    report_progress()
    set_digital_out(0, False)
    new_pose = pose_trans(tuft_coords, p[1.0096, 0.7853, 0.1500, 0, 0, 0])
    movel(p[new_pose[0], new_pose[1], new_pose[2], current_pose[3], current_pose[4], current_pose[5]], a=0.8, v=0.2000)
    report_progress()
    new_pose = pose_trans(tuft_coords, p[1.0115, 0.2667, 0.1500, 0, 0, 0])
    movel(p[new_pose[0], new_pose[1], new_pose[2], current_pose[3], current_pose[4], current_pose[5]], a=1.2, v=0.2000)
    report_progress()
    new_pose = pose_trans(tuft_coords, p[1.0115, 0.2667, -0.0020, 0, 0, 0])
    movel(p[new_pose[0], new_pose[1], new_pose[2], current_pose[3], current_pose[4], current_pose[5]], a=0.8, v=0.2000)
    report_progress()
    set_digital_out(0, True)
    new_pose = pose_trans(tuft_coords, p[1.0115, 0.7833, -0.0020, 0, 0, 0])
    movel(p[new_pose[0], new_pose[1], new_pose[2], current_pose[3], current_pose[4], current_pose[5]], a=1.2, v=0.0600)
    report_progress()
    set_digital_out(0, False)
    new_pose = pose_trans(tuft_coords, p[1.0115, 0.7833, 0.1500, 0, 0, 0])
    movel(p[new_pose[0], new_pose[1], new_pose[2], current_pose[3], current_pose[4], current_pose[5]], a=0.8, v=0.2000)
    report_progress()
    new_pose = pose_trans(tuft_coords, p[1.0135, 0.2687, 0.1500, 0, 0, 0])
    movel(p[new_pose[0], new_pose[1], new_pose[2], current_pose[3], current_pose[4], current_pose[5]], a=1.2, v=0.2000)
    report_progress()
    new_pose = pose_trans(tuft_coords, p[1.0135, 0.2687, -0.0020, 0, 0, 0])
    movel(p[new_pose[0], new_pose[1], new_pose[2], current_pose[3], current_pose[4], current_pose[5]], a=0.8, v=0.2000)
    report_progress()
    set_digital_out(0, True)
    new_pose = pose_trans(tuft_coords, p[1.0135, 0.7813, -0.0020, 0, 0, 0])
    movel(p[new_pose[0], new_pose[1], new_pose[2], current_pose[3], current_pose[4], current_pose[5]], a=1.2, v=0.0600)
    report_progress()
    set_digital_out(0, False)
    new_pose = pose_trans(tuft_coords, p[1.0135, 0.7813, 0.1500, 0, 0, 0])
    movel(p[new_pose[0], new_pose[1], new_pose[2], current_pose[3], current_pose[4], current_pose[5]], a=0.8, v=0.2000)
    report_progress()
    new_pose = pose_trans(tuft_coords, p[1.0154, 0.2707, 0.1500, 0, 0, 0])
    movel(p[new_pose[0], new_pose[1], new_pose[2], current_pose[3], current_pose[4], current_pose[5]], a=1.2, v=0.2000)
    report_progress()
    new_pose = pose_trans(tuft_coords, p[1.0154, 0.2707, -0.0020, 0, 0, 0])
    movel(p[new_pose[0], new_pose[1], new_pose[2], current_pose[3], current_pose[4], current_pose[5]], a=0.8, v=0.2000)
    report_progress()
    set_digital_out(0, True)
    new_pose = pose_trans(tuft_coords, p[1.0154, 0.7793, -0.0020, 0, 0, 0])
    movel(p[new_pose[0], new_pose[1], new_pose[2], current_pose[3], current_pose[4], current_pose[5]], a=1.2, v=0.0600)
    report_progress()
    set_digital_out(0, False)
    new_pose = pose_trans(tuft_coords, p[1.0154, 0.7793, 0.1500, 0, 0, 0])
    movel(p[new_pose[0], new_pose[1], new_pose[2], current_pose[3], current_pose[4], current_pose[5]], a=0.8, v=0.2000)
    report_progress()
    new_pose = pose_trans(tuft_coords, p[1.0174, 0.2727, 0.1500, 0, 0, 0])
    movel(p[new_pose[0], new_pose[1], new_pose[2], current_pose[3], current_pose[4], current_pose[5]], a=1.2, v=0.2000)
    report_progress()
    new_pose = pose_trans(tuft_coords, p[1.0174, 0.2727, -0.0020, 0, 0, 0])
    movel(p[new_pose[0], new_pose[1], new_pose[2], current_pose[3], current_pose[4], current_pose[5]], a=0.8, v=0.2000)
    report_progress()
    set_digital_out(0, True)
    new_pose = pose_trans(tuft_coords, p[1.0174, 0.7773, -0.0020, 0, 0, 0])
    movel(p[new_pose[0], new_pose[1], new_pose[2], current_pose[3], current_pose[4], current_pose[5]], a=1.2, v=0.0600)
    report_progress()
    set_digital_out(0, False)
    new_pose = pose_trans(tuft_coords, p[1.0174, 0.7773, 0.1500, 0, 0, 0])
    movel(p[new_pose[0], new_pose[1], new_pose[2], current_pose[3], current_pose[4], current_pose[5]], a=0.8, v=0.2000)
    report_progress()
    new_pose = pose_trans(tuft_coords, p[1.0193, 0.2746, 0.1500, 0, 0, 0])
    movel(p[new_pose[0], new_pose[1], new_pose[2], current_pose[3], current_pose[4], current_pose[5]], a=1.2, v=0.2000)
    report_progress()
    new_pose = pose_trans(tuft_coords, p[1.0193, 0.2746, -0.0020, 0, 0, 0])
    movel(p[new_pose[0], new_pose[1], new_pose[2], current_pose[3], current_pose[4], current_pose[5]], a=0.8, v=0.2000)
    report_progress()
    set_digital_out(0, True)
    new_pose = pose_trans(tuft_coords, p[1.0193, 0.7754, -0.0020, 0, 0, 0])
    movel(p[new_pose[0], new_pose[1], new_pose[2], current_pose[3], current_pose[4], current_pose[5]], a=1.2, v=0.0600)
    report_progress()
    set_digital_out(0, False)
    new_pose = pose_trans(tuft_coords, p[1.0193, 0.7754, 0.1500, 0, 0, 0])
    movel(p[new_pose[0], new_pose[1], new_pose[2], current_pose[3], current_pose[4], current_pose[5]], a=0.8, v=0.2000)
    report_progress()
    new_pose = pose_trans(tuft_coords, p[1.0212, 0.2766, 0.1500, 0, 0, 0])
    movel(p[new_pose[0], new_pose[1], new_pose[2], current_pose[3], current_pose[4], current_pose[5]], a=1.2, v=0.2000)
    report_progress()
    new_pose = pose_trans(tuft_coords, p[1.0212, 0.2766, -0.0020, 0, 0, 0])
    movel(p[new_pose[0], new_pose[1], new_pose[2], current_pose[3], current_pose[4], current_pose[5]], a=0.8, v=0.2000)
    report_progress()
    set_digital_out(0, True)
    new_pose = pose_trans(tuft_coords, p[1.0212, 0.7734, -0.0020, 0, 0, 0])
    movel(p[new_pose[0], new_pose[1], new_pose[2], current_pose[3], current_pose[4], current_pose[5]], a=1.2, v=0.0600)
    report_progress()
    set_digital_out(0, False)
    new_pose = pose_trans(tuft_coords, p[1.0212, 0.7734, 0.1500, 0, 0, 0])
    movel(p[new_pose[0], new_pose[1], new_pose[2], current_pose[3], current_pose[4], current_pose[5]], a=0.8, v=0.2000)
    report_progress()
    new_pose = pose_trans(tuft_coords, p[1.0232, 0.2786, 0.1500, 0, 0, 0])
    movel(p[new_pose[0], new_pose[1], new_pose[2], current_pose[3], current_pose[4], current_pose[5]], a=1.2, v=0.2000)
    report_progress()
    new_pose = pose_trans(tuft_coords, p[1.0232, 0.2786, -0.0020, 0, 0, 0])
    movel(p[new_pose[0], new_pose[1], new_pose[2], current_pose[3], current_pose[4], current_pose[5]], a=0.8, v=0.2000)
    report_progress()
    set_digital_out(0, True)
    new_pose = pose_trans(tuft_coords, p[1.0232, 0.7714, -0.0020, 0, 0, 0])
    movel(p[new_pose[0], new_pose[1], new_pose[2], current_pose[3], current_pose[4], current_pose[5]], a=1.2, v=0.0600)
    report_progress()
    set_digital_out(0, False)
    new_pose = pose_trans(tuft_coords, p[1.0232, 0.7714, 0.1500, 0, 0, 0])
    movel(p[new_pose[0], new_pose[1], new_pose[2], current_pose[3], current_pose[4], current_pose[5]], a=0.8, v=0.2000)
    report_progress()
    new_pose = pose_trans(tuft_coords, p[1.0251, 0.2826, 0.1500, 0, 0, 0])
    movel(p[new_pose[0], new_pose[1], new_pose[2], current_pose[3], current_pose[4], current_pose[5]], a=1.2, v=0.2000)
    report_progress()
    new_pose = pose_trans(tuft_coords, p[1.0251, 0.2826, -0.0020, 0, 0, 0])
    movel(p[new_pose[0], new_pose[1], new_pose[2], current_pose[3], current_pose[4], current_pose[5]], a=0.8, v=0.2000)
    report_progress()
    set_digital_out(0, True)
    new_pose = pose_trans(tuft_coords, p[1.0251, 0.7674, -0.0020, 0, 0, 0])
    movel(p[new_pose[0], new_pose[1], new_pose[2], current_pose[3], current_pose[4], current_pose[5]], a=1.2, v=0.0600)
    report_progress()
    set_digital_out(0, False)
    new_pose = pose_trans(tuft_coords, p[1.0251, 0.7674, 0.1500, 0, 0, 0])
    movel(p[new_pose[0], new_pose[1], new_pose[2], current_pose[3], current_pose[4], current_pose[5]], a=0.8, v=0.2000)
    report_progress()
    new_pose = pose_trans(tuft_coords, p[1.0271, 0.2845, 0.1500, 0, 0, 0])
    movel(p[new_pose[0], new_pose[1], new_pose[2], current_pose[3], current_pose[4], current_pose[5]], a=1.2, v=0.2000)
    report_progress()
    new_pose = pose_trans(tuft_coords, p[1.0271, 0.2845, -0.0020, 0, 0, 0])
    movel(p[new_pose[0], new_pose[1], new_pose[2], current_pose[3], current_pose[4], current_pose[5]], a=0.8, v=0.2000)
    report_progress()
    set_digital_out(0, True)
    new_pose = pose_trans(tuft_coords, p[1.0271, 0.7655, -0.0020, 0, 0, 0])
    movel(p[new_pose[0], new_pose[1], new_pose[2], current_pose[3], current_pose[4], current_pose[5]], a=1.2, v=0.0600)
    report_progress()
    set_digital_out(0, False)
    new_pose = pose_trans(tuft_coords, p[1.0271, 0.7655, 0.1500, 0, 0, 0])
    movel(p[new_pose[0], new_pose[1], new_pose[2], current_pose[3], current_pose[4], current_pose[5]], a=0.8, v=0.2000)
    report_progress()
    new_pose = pose_trans(tuft_coords, p[1.0290, 0.2865, 0.1500, 0, 0, 0])
    movel(p[new_pose[0], new_pose[1], new_pose[2], current_pose[3], current_pose[4], current_pose[5]], a=1.2, v=0.2000)
    report_progress()
    new_pose = pose_trans(tuft_coords, p[1.0290, 0.2865, -0.0020, 0, 0, 0])
    movel(p[new_pose[0], new_pose[1], new_pose[2], current_pose[3], current_pose[4], current_pose[5]], a=0.8, v=0.2000)
    report_progress()
    set_digital_out(0, True)
    new_pose = pose_trans(tuft_coords, p[1.0290, 0.7635, -0.0020, 0, 0, 0])
    movel(p[new_pose[0], new_pose[1], new_pose[2], current_pose[3], current_pose[4], current_pose[5]], a=1.2, v=0.0600)
    report_progress()
    set_digital_out(0, False)
    new_pose = pose_trans(tuft_coords, p[1.0290, 0.7635, 0.1500, 0, 0, 0])
    movel(p[new_pose[0], new_pose[1], new_pose[2], current_pose[3], current_pose[4], current_pose[5]], a=0.8, v=0.2000)
    report_progress()
    new_pose = pose_trans(tuft_coords, p[1.0310, 0.2885, 0.1500, 0, 0, 0])
    movel(p[new_pose[0], new_pose[1], new_pose[2], current_pose[3], current_pose[4], current_pose[5]], a=1.2, v=0.2000)
    report_progress()
    new_pose = pose_trans(tuft_coords, p[1.0310, 0.2885, -0.0020, 0, 0, 0])
    movel(p[new_pose[0], new_pose[1], new_pose[2], current_pose[3], current_pose[4], current_pose[5]], a=0.8, v=0.2000)
    report_progress()
    set_digital_out(0, True)
    new_pose = pose_trans(tuft_coords, p[1.0310, 0.7615, -0.0020, 0, 0, 0])
    movel(p[new_pose[0], new_pose[1], new_pose[2], current_pose[3], current_pose[4], current_pose[5]], a=1.2, v=0.0600)
    report_progress()
    set_digital_out(0, False)
    new_pose = pose_trans(tuft_coords, p[1.0310, 0.7615, 0.1500, 0, 0, 0])
    movel(p[new_pose[0], new_pose[1], new_pose[2], current_pose[3], current_pose[4], current_pose[5]], a=0.8, v=0.2000)
    report_progress()
    new_pose = pose_trans(tuft_coords, p[1.0329, 0.2905, 0.1500, 0, 0, 0])
    movel(p[new_pose[0], new_pose[1], new_pose[2], current_pose[3], current_pose[4], current_pose[5]], a=1.2, v=0.2000)
    report_progress()
    new_pose = pose_trans(tuft_coords, p[1.0329, 0.2905, -0.0020, 0, 0, 0])
    movel(p[new_pose[0], new_pose[1], new_pose[2], current_pose[3], current_pose[4], current_pose[5]], a=0.8, v=0.2000)
    report_progress()
    set_digital_out(0, True)
    new_pose = pose_trans(tuft_coords, p[1.0329, 0.7595, -0.0020, 0, 0, 0])
    movel(p[new_pose[0], new_pose[1], new_pose[2], current_pose[3], current_pose[4], current_pose[5]], a=1.2, v=0.0600)
    report_progress()
    set_digital_out(0, False)
    new_pose = pose_trans(tuft_coords, p[1.0329, 0.7595, 0.1500, 0, 0, 0])
    movel(p[new_pose[0], new_pose[1], new_pose[2], current_pose[3], current_pose[4], current_pose[5]], a=0.8, v=0.2000)
    report_progress()
    new_pose = pose_trans(tuft_coords, p[1.0349, 0.2944, 0.1500, 0, 0, 0])
    movel(p[new_pose[0], new_pose[1], new_pose[2], current_pose[3], current_pose[4], current_pose[5]], a=1.2, v=0.2000)
    report_progress()
    new_pose = pose_trans(tuft_coords, p[1.0349, 0.2944, -0.0020, 0, 0, 0])
    movel(p[new_pose[0], new_pose[1], new_pose[2], current_pose[3], current_pose[4], current_pose[5]], a=0.8, v=0.2000)
    report_progress()
    set_digital_out(0, True)
    new_pose = pose_trans(tuft_coords, p[1.0349, 0.7556, -0.0020, 0, 0, 0])
    movel(p[new_pose[0], new_pose[1], new_pose[2], current_pose[3], current_pose[4], current_pose[5]], a=1.2, v=0.0600)
    report_progress()
    set_digital_out(0, False)
    new_pose = pose_trans(tuft_coords, p[1.0349, 0.7556, 0.1500, 0, 0, 0])
    movel(p[new_pose[0], new_pose[1], new_pose[2], current_pose[3], current_pose[4], current_pose[5]], a=0.8, v=0.2000)
    report_progress()
    new_pose = pose_trans(tuft_coords, p[1.0368, 0.2964, 0.1500, 0, 0, 0])
    movel(p[new_pose[0], new_pose[1], new_pose[2], current_pose[3], current_pose[4], current_pose[5]], a=1.2, v=0.2000)
    report_progress()
    new_pose = pose_trans(tuft_coords, p[1.0368, 0.2964, -0.0020, 0, 0, 0])
    movel(p[new_pose[0], new_pose[1], new_pose[2], current_pose[3], current_pose[4], current_pose[5]], a=0.8, v=0.2000)
    report_progress()
    set_digital_out(0, True)
    new_pose = pose_trans(tuft_coords, p[1.0368, 0.7536, -0.0020, 0, 0, 0])
    movel(p[new_pose[0], new_pose[1], new_pose[2], current_pose[3], current_pose[4], current_pose[5]], a=1.2, v=0.0600)
    report_progress()
    set_digital_out(0, False)
    new_pose = pose_trans(tuft_coords, p[1.0368, 0.7536, 0.1500, 0, 0, 0])
    movel(p[new_pose[0], new_pose[1], new_pose[2], current_pose[3], current_pose[4], current_pose[5]], a=0.8, v=0.2000)
    report_progress()
    new_pose = pose_trans(tuft_coords, p[1.0388, 0.2984, 0.1500, 0, 0, 0])
    movel(p[new_pose[0], new_pose[1], new_pose[2], current_pose[3], current_pose[4], current_pose[5]], a=1.2, v=0.2000)
    report_progress()
    new_pose = pose_trans(tuft_coords, p[1.0388, 0.2984, -0.0020, 0, 0, 0])
    movel(p[new_pose[0], new_pose[1], new_pose[2], current_pose[3], current_pose[4], current_pose[5]], a=0.8, v=0.2000)
    report_progress()
    set_digital_out(0, True)
    new_pose = pose_trans(tuft_coords, p[1.0388, 0.7516, -0.0020, 0, 0, 0])
    movel(p[new_pose[0], new_pose[1], new_pose[2], current_pose[3], current_pose[4], current_pose[5]], a=1.2, v=0.0600)
    report_progress()
    set_digital_out(0, False)
    new_pose = pose_trans(tuft_coords, p[1.0388, 0.7516, 0.1500, 0, 0, 0])
    movel(p[new_pose[0], new_pose[1], new_pose[2], current_pose[3], current_pose[4], current_pose[5]], a=0.8, v=0.2000)
    report_progress()
    new_pose = pose_trans(tuft_coords, p[1.0407, 0.3004, 0.1500, 0, 0, 0])
    movel(p[new_pose[0], new_pose[1], new_pose[2], current_pose[3], current_pose[4], current_pose[5]], a=1.2, v=0.2000)
    report_progress()
    new_pose = pose_trans(tuft_coords, p[1.0407, 0.3004, -0.0020, 0, 0, 0])
    movel(p[new_pose[0], new_pose[1], new_pose[2], current_pose[3], current_pose[4], current_pose[5]], a=0.8, v=0.2000)
    report_progress()
    set_digital_out(0, True)
    new_pose = pose_trans(tuft_coords, p[1.0407, 0.7496, -0.0020, 0, 0, 0])
    movel(p[new_pose[0], new_pose[1], new_pose[2], current_pose[3], current_pose[4], current_pose[5]], a=1.2, v=0.0600)
    report_progress()
    set_digital_out(0, False)
    new_pose = pose_trans(tuft_coords, p[1.0407, 0.7496, 0.1500, 0, 0, 0])
    movel(p[new_pose[0], new_pose[1], new_pose[2], current_pose[3], current_pose[4], current_pose[5]], a=0.8, v=0.2000)
    report_progress()
    new_pose = pose_trans(tuft_coords, p[1.0426, 0.3043, 0.1500, 0, 0, 0])
    movel(p[new_pose[0], new_pose[1], new_pose[2], current_pose[3], current_pose[4], current_pose[5]], a=1.2, v=0.2000)
    report_progress()
    new_pose = pose_trans(tuft_coords, p[1.0426, 0.3043, -0.0020, 0, 0, 0])
    movel(p[new_pose[0], new_pose[1], new_pose[2], current_pose[3], current_pose[4], current_pose[5]], a=0.8, v=0.2000)
    report_progress()
    set_digital_out(0, True)
    new_pose = pose_trans(tuft_coords, p[1.0426, 0.7457, -0.0020, 0, 0, 0])
    movel(p[new_pose[0], new_pose[1], new_pose[2], current_pose[3], current_pose[4], current_pose[5]], a=1.2, v=0.0600)
    report_progress()
    set_digital_out(0, False)
    new_pose = pose_trans(tuft_coords, p[1.0426, 0.7457, 0.1500, 0, 0, 0])
    movel(p[new_pose[0], new_pose[1], new_pose[2], current_pose[3], current_pose[4], current_pose[5]], a=0.8, v=0.2000)
    report_progress()
    new_pose = pose_trans(tuft_coords, p[1.0446, 0.3063, 0.1500, 0, 0, 0])
    movel(p[new_pose[0], new_pose[1], new_pose[2], current_pose[3], current_pose[4], current_pose[5]], a=1.2, v=0.2000)
    report_progress()
    new_pose = pose_trans(tuft_coords, p[1.0446, 0.3063, -0.0020, 0, 0, 0])
    movel(p[new_pose[0], new_pose[1], new_pose[2], current_pose[3], current_pose[4], current_pose[5]], a=0.8, v=0.2000)
    report_progress()
    set_digital_out(0, True)
    new_pose = pose_trans(tuft_coords, p[1.0446, 0.7437, -0.0020, 0, 0, 0])
    movel(p[new_pose[0], new_pose[1], new_pose[2], current_pose[3], current_pose[4], current_pose[5]], a=1.2, v=0.0600)
    report_progress()
    set_digital_out(0, False)
    new_pose = pose_trans(tuft_coords, p[1.0446, 0.7437, 0.1500, 0, 0, 0])
    movel(p[new_pose[0], new_pose[1], new_pose[2], current_pose[3], current_pose[4], current_pose[5]], a=0.8, v=0.2000)
    report_progress()
    new_pose = pose_trans(tuft_coords, p[1.0465, 0.3083, 0.1500, 0, 0, 0])
    movel(p[new_pose[0], new_pose[1], new_pose[2], current_pose[3], current_pose[4], current_pose[5]], a=1.2, v=0.2000)
    report_progress()
    new_pose = pose_trans(tuft_coords, p[1.0465, 0.3083, -0.0020, 0, 0, 0])
    movel(p[new_pose[0], new_pose[1], new_pose[2], current_pose[3], current_pose[4], current_pose[5]], a=0.8, v=0.2000)
    report_progress()
    set_digital_out(0, True)
    new_pose = pose_trans(tuft_coords, p[1.0465, 0.7417, -0.0020, 0, 0, 0])
    movel(p[new_pose[0], new_pose[1], new_pose[2], current_pose[3], current_pose[4], current_pose[5]], a=1.2, v=0.0600)
    report_progress()
    set_digital_out(0, False)
    new_pose = pose_trans(tuft_coords, p[1.0465, 0.7417, 0.1500, 0, 0, 0])
    movel(p[new_pose[0], new_pose[1], new_pose[2], current_pose[3], current_pose[4], current_pose[5]], a=0.8, v=0.2000)
    report_progress()
    new_pose = pose_trans(tuft_coords, p[1.0485, 0.3122, 0.1500, 0, 0, 0])
    movel(p[new_pose[0], new_pose[1], new_pose[2], current_pose[3], current_pose[4], current_pose[5]], a=1.2, v=0.2000)
    report_progress()
    new_pose = pose_trans(tuft_coords, p[1.0485, 0.3122, -0.0020, 0, 0, 0])
    movel(p[new_pose[0], new_pose[1], new_pose[2], current_pose[3], current_pose[4], current_pose[5]], a=0.8, v=0.2000)
    report_progress()
    set_digital_out(0, True)
    new_pose = pose_trans(tuft_coords, p[1.0485, 0.7378, -0.0020, 0, 0, 0])
    movel(p[new_pose[0], new_pose[1], new_pose[2], current_pose[3], current_pose[4], current_pose[5]], a=1.2, v=0.0600)
    report_progress()
    set_digital_out(0, False)
    new_pose = pose_trans(tuft_coords, p[1.0485, 0.7378, 0.1500, 0, 0, 0])
    movel(p[new_pose[0], new_pose[1], new_pose[2], current_pose[3], current_pose[4], current_pose[5]], a=0.8, v=0.2000)
    report_progress()
    new_pose = pose_trans(tuft_coords, p[1.0504, 0.3142, 0.1500, 0, 0, 0])
    movel(p[new_pose[0], new_pose[1], new_pose[2], current_pose[3], current_pose[4], current_pose[5]], a=1.2, v=0.2000)
    report_progress()
    new_pose = pose_trans(tuft_coords, p[1.0504, 0.3142, -0.0020, 0, 0, 0])
    movel(p[new_pose[0], new_pose[1], new_pose[2], current_pose[3], current_pose[4], current_pose[5]], a=0.8, v=0.2000)
    report_progress()
    set_digital_out(0, True)
    new_pose = pose_trans(tuft_coords, p[1.0504, 0.7358, -0.0020, 0, 0, 0])
    movel(p[new_pose[0], new_pose[1], new_pose[2], current_pose[3], current_pose[4], current_pose[5]], a=1.2, v=0.0600)
    report_progress()
    set_digital_out(0, False)
    new_pose = pose_trans(tuft_coords, p[1.0504, 0.7358, 0.1500, 0, 0, 0])
    movel(p[new_pose[0], new_pose[1], new_pose[2], current_pose[3], current_pose[4], current_pose[5]], a=0.8, v=0.2000)
    report_progress()
    new_pose = pose_trans(tuft_coords, p[1.0524, 0.3182, 0.1500, 0, 0, 0])
    movel(p[new_pose[0], new_pose[1], new_pose[2], current_pose[3], current_pose[4], current_pose[5]], a=1.2, v=0.2000)
    report_progress()
    new_pose = pose_trans(tuft_coords, p[1.0524, 0.3182, -0.0020, 0, 0, 0])
    movel(p[new_pose[0], new_pose[1], new_pose[2], current_pose[3], current_pose[4], current_pose[5]], a=0.8, v=0.2000)
    report_progress()
    set_digital_out(0, True)
    new_pose = pose_trans(tuft_coords, p[1.0524, 0.7318, -0.0020, 0, 0, 0])
    movel(p[new_pose[0], new_pose[1], new_pose[2], current_pose[3], current_pose[4], current_pose[5]], a=1.2, v=0.0600)
    report_progress()
    set_digital_out(0, False)
    new_pose = pose_trans(tuft_coords, p[1.0524, 0.7318, 0.1500, 0, 0, 0])
    movel(p[new_pose[0], new_pose[1], new_pose[2], current_pose[3], current_pose[4], current_pose[5]], a=0.8, v=0.2000)
    report_progress()
    new_pose = pose_trans(tuft_coords, p[1.0543, 0.3202, 0.1500, 0, 0, 0])
    movel(p[new_pose[0], new_pose[1], new_pose[2], current_pose[3], current_pose[4], current_pose[5]], a=1.2, v=0.2000)
    report_progress()
    new_pose = pose_trans(tuft_coords, p[1.0543, 0.3202, -0.0020, 0, 0, 0])
    movel(p[new_pose[0], new_pose[1], new_pose[2], current_pose[3], current_pose[4], current_pose[5]], a=0.8, v=0.2000)
    report_progress()
    set_digital_out(0, True)
    new_pose = pose_trans(tuft_coords, p[1.0543, 0.7298, -0.0020, 0, 0, 0])
    movel(p[new_pose[0], new_pose[1], new_pose[2], current_pose[3], current_pose[4], current_pose[5]], a=1.2, v=0.0600)
    report_progress()
    set_digital_out(0, False)
    new_pose = pose_trans(tuft_coords, p[1.0543, 0.7298, 0.1500, 0, 0, 0])
    movel(p[new_pose[0], new_pose[1], new_pose[2], current_pose[3], current_pose[4], current_pose[5]], a=0.8, v=0.2000)
    report_progress()
    new_pose = pose_trans(tuft_coords, p[1.0562, 0.3241, 0.1500, 0, 0, 0])
    movel(p[new_pose[0], new_pose[1], new_pose[2], current_pose[3], current_pose[4], current_pose[5]], a=1.2, v=0.2000)
    report_progress()
    new_pose = pose_trans(tuft_coords, p[1.0562, 0.3241, -0.0020, 0, 0, 0])
    movel(p[new_pose[0], new_pose[1], new_pose[2], current_pose[3], current_pose[4], current_pose[5]], a=0.8, v=0.2000)
    report_progress()
    set_digital_out(0, True)
    new_pose = pose_trans(tuft_coords, p[1.0562, 0.7259, -0.0020, 0, 0, 0])
    movel(p[new_pose[0], new_pose[1], new_pose[2], current_pose[3], current_pose[4], current_pose[5]], a=1.2, v=0.0600)
    report_progress()
    set_digital_out(0, False)
    new_pose = pose_trans(tuft_coords, p[1.0562, 0.7259, 0.1500, 0, 0, 0])
    movel(p[new_pose[0], new_pose[1], new_pose[2], current_pose[3], current_pose[4], current_pose[5]], a=0.8, v=0.2000)
    report_progress()
    new_pose = pose_trans(tuft_coords, p[1.0582, 0.3261, 0.1500, 0, 0, 0])
    movel(p[new_pose[0], new_pose[1], new_pose[2], current_pose[3], current_pose[4], current_pose[5]], a=1.2, v=0.2000)
    report_progress()
    new_pose = pose_trans(tuft_coords, p[1.0582, 0.3261, -0.0020, 0, 0, 0])
    movel(p[new_pose[0], new_pose[1], new_pose[2], current_pose[3], current_pose[4], current_pose[5]], a=0.8, v=0.2000)
    report_progress()
    set_digital_out(0, True)
    new_pose = pose_trans(tuft_coords, p[1.0582, 0.7239, -0.0020, 0, 0, 0])
    movel(p[new_pose[0], new_pose[1], new_pose[2], current_pose[3], current_pose[4], current_pose[5]], a=1.2, v=0.0600)
    report_progress()
    set_digital_out(0, False)
    new_pose = pose_trans(tuft_coords, p[1.0582, 0.7239, 0.1500, 0, 0, 0])
    movel(p[new_pose[0], new_pose[1], new_pose[2], current_pose[3], current_pose[4], current_pose[5]], a=0.8, v=0.2000)
    report_progress()
    new_pose = pose_trans(tuft_coords, p[1.0601, 0.3301, 0.1500, 0, 0, 0])
    movel(p[new_pose[0], new_pose[1], new_pose[2], current_pose[3], current_pose[4], current_pose[5]], a=1.2, v=0.2000)
    report_progress()
    new_pose = pose_trans(tuft_coords, p[1.0601, 0.3301, -0.0020, 0, 0, 0])
    movel(p[new_pose[0], new_pose[1], new_pose[2], current_pose[3], current_pose[4], current_pose[5]], a=0.8, v=0.2000)
    report_progress()
    set_digital_out(0, True)
    new_pose = pose_trans(tuft_coords, p[1.0601, 0.7199, -0.0020, 0, 0, 0])
    movel(p[new_pose[0], new_pose[1], new_pose[2], current_pose[3], current_pose[4], current_pose[5]], a=1.2, v=0.0600)
    report_progress()
    set_digital_out(0, False)
    new_pose = pose_trans(tuft_coords, p[1.0601, 0.7199, 0.1500, 0, 0, 0])
    movel(p[new_pose[0], new_pose[1], new_pose[2], current_pose[3], current_pose[4], current_pose[5]], a=0.8, v=0.2000)
    report_progress()
    new_pose = pose_trans(tuft_coords, p[1.0621, 0.3340, 0.1500, 0, 0, 0])
    movel(p[new_pose[0], new_pose[1], new_pose[2], current_pose[3], current_pose[4], current_pose[5]], a=1.2, v=0.2000)
    report_progress()
    new_pose = pose_trans(tuft_coords, p[1.0621, 0.3340, -0.0020, 0, 0, 0])
    movel(p[new_pose[0], new_pose[1], new_pose[2], current_pose[3], current_pose[4], current_pose[5]], a=0.8, v=0.2000)
    report_progress()
    set_digital_out(0, True)
    new_pose = pose_trans(tuft_coords, p[1.0621, 0.7160, -0.0020, 0, 0, 0])
    movel(p[new_pose[0], new_pose[1], new_pose[2], current_pose[3], current_pose[4], current_pose[5]], a=1.2, v=0.0600)
    report_progress()
    set_digital_out(0, False)
    new_pose = pose_trans(tuft_coords, p[1.0621, 0.7160, 0.1500, 0, 0, 0])
    movel(p[new_pose[0], new_pose[1], new_pose[2], current_pose[3], current_pose[4], current_pose[5]], a=0.8, v=0.2000)
    report_progress()
    new_pose = pose_trans(tuft_coords, p[1.0640, 0.3360, 0.1500, 0, 0, 0])
    movel(p[new_pose[0], new_pose[1], new_pose[2], current_pose[3], current_pose[4], current_pose[5]], a=1.2, v=0.2000)
    report_progress()
    new_pose = pose_trans(tuft_coords, p[1.0640, 0.3360, -0.0020, 0, 0, 0])
    movel(p[new_pose[0], new_pose[1], new_pose[2], current_pose[3], current_pose[4], current_pose[5]], a=0.8, v=0.2000)
    report_progress()
    set_digital_out(0, True)
    new_pose = pose_trans(tuft_coords, p[1.0640, 0.7140, -0.0020, 0, 0, 0])
    movel(p[new_pose[0], new_pose[1], new_pose[2], current_pose[3], current_pose[4], current_pose[5]], a=1.2, v=0.0600)
    report_progress()
    set_digital_out(0, False)
    new_pose = pose_trans(tuft_coords, p[1.0640, 0.7140, 0.1500, 0, 0, 0])
    movel(p[new_pose[0], new_pose[1], new_pose[2], current_pose[3], current_pose[4], current_pose[5]], a=0.8, v=0.2000)
    report_progress()
    new_pose = pose_trans(tuft_coords, p[1.0660, 0.3399, 0.1500, 0, 0, 0])
    movel(p[new_pose[0], new_pose[1], new_pose[2], current_pose[3], current_pose[4], current_pose[5]], a=1.2, v=0.2000)
    report_progress()
    new_pose = pose_trans(tuft_coords, p[1.0660, 0.3399, -0.0020, 0, 0, 0])
    movel(p[new_pose[0], new_pose[1], new_pose[2], current_pose[3], current_pose[4], current_pose[5]], a=0.8, v=0.2000)
    report_progress()
    set_digital_out(0, True)
    new_pose = pose_trans(tuft_coords, p[1.0660, 0.7101, -0.0020, 0, 0, 0])
    movel(p[new_pose[0], new_pose[1], new_pose[2], current_pose[3], current_pose[4], current_pose[5]], a=1.2, v=0.0600)
    report_progress()
    set_digital_out(0, False)
    new_pose = pose_trans(tuft_coords, p[1.0660, 0.7101, 0.1500, 0, 0, 0])
    movel(p[new_pose[0], new_pose[1], new_pose[2], current_pose[3], current_pose[4], current_pose[5]], a=0.8, v=0.2000)
    report_progress()
    new_pose = pose_trans(tuft_coords, p[1.0679, 0.3439, 0.1500, 0, 0, 0])
    movel(p[new_pose[0], new_pose[1], new_pose[2], current_pose[3], current_pose[4], current_pose[5]], a=1.2, v=0.2000)
    report_progress()
    new_pose = pose_trans(tuft_coords, p[1.0679, 0.3439, -0.0020, 0, 0, 0])
    movel(p[new_pose[0], new_pose[1], new_pose[2], current_pose[3], current_pose[4], current_pose[5]], a=0.8, v=0.2000)
    report_progress()
    set_digital_out(0, True)
    new_pose = pose_trans(tuft_coords, p[1.0679, 0.7061, -0.0020, 0, 0, 0])
    movel(p[new_pose[0], new_pose[1], new_pose[2], current_pose[3], current_pose[4], current_pose[5]], a=1.2, v=0.0600)
    report_progress()
    set_digital_out(0, False)
    new_pose = pose_trans(tuft_coords, p[1.0679, 0.7061, 0.1500, 0, 0, 0])
    movel(p[new_pose[0], new_pose[1], new_pose[2], current_pose[3], current_pose[4], current_pose[5]], a=0.8, v=0.2000)
    report_progress()
    new_pose = pose_trans(tuft_coords, p[1.0699, 0.3459, 0.1500, 0, 0, 0])
    movel(p[new_pose[0], new_pose[1], new_pose[2], current_pose[3], current_pose[4], current_pose[5]], a=1.2, v=0.2000)
    report_progress()
    new_pose = pose_trans(tuft_coords, p[1.0699, 0.3459, -0.0020, 0, 0, 0])
    movel(p[new_pose[0], new_pose[1], new_pose[2], current_pose[3], current_pose[4], current_pose[5]], a=0.8, v=0.2000)
    report_progress()
    set_digital_out(0, True)
    new_pose = pose_trans(tuft_coords, p[1.0699, 0.7041, -0.0020, 0, 0, 0])
    movel(p[new_pose[0], new_pose[1], new_pose[2], current_pose[3], current_pose[4], current_pose[5]], a=1.2, v=0.0600)
    report_progress()
    set_digital_out(0, False)
    new_pose = pose_trans(tuft_coords, p[1.0699, 0.7041, 0.1500, 0, 0, 0])
    movel(p[new_pose[0], new_pose[1], new_pose[2], current_pose[3], current_pose[4], current_pose[5]], a=0.8, v=0.2000)
    report_progress()
    new_pose = pose_trans(tuft_coords, p[1.0718, 0.3498, 0.1500, 0, 0, 0])
    movel(p[new_pose[0], new_pose[1], new_pose[2], current_pose[3], current_pose[4], current_pose[5]], a=1.2, v=0.2000)
    report_progress()
    new_pose = pose_trans(tuft_coords, p[1.0718, 0.3498, -0.0020, 0, 0, 0])
    movel(p[new_pose[0], new_pose[1], new_pose[2], current_pose[3], current_pose[4], current_pose[5]], a=0.8, v=0.2000)
    report_progress()
    set_digital_out(0, True)
    new_pose = pose_trans(tuft_coords, p[1.0718, 0.7002, -0.0020, 0, 0, 0])
    movel(p[new_pose[0], new_pose[1], new_pose[2], current_pose[3], current_pose[4], current_pose[5]], a=1.2, v=0.0600)
    report_progress()
    set_digital_out(0, False)
    new_pose = pose_trans(tuft_coords, p[1.0718, 0.7002, 0.1500, 0, 0, 0])
    movel(p[new_pose[0], new_pose[1], new_pose[2], current_pose[3], current_pose[4], current_pose[5]], a=0.8, v=0.2000)
    report_progress()
    new_pose = pose_trans(tuft_coords, p[1.0737, 0.3538, 0.1500, 0, 0, 0])
    movel(p[new_pose[0], new_pose[1], new_pose[2], current_pose[3], current_pose[4], current_pose[5]], a=1.2, v=0.2000)
    report_progress()
    new_pose = pose_trans(tuft_coords, p[1.0737, 0.3538, -0.0020, 0, 0, 0])
    movel(p[new_pose[0], new_pose[1], new_pose[2], current_pose[3], current_pose[4], current_pose[5]], a=0.8, v=0.2000)
    report_progress()
    set_digital_out(0, True)
    new_pose = pose_trans(tuft_coords, p[1.0737, 0.6962, -0.0020, 0, 0, 0])
    movel(p[new_pose[0], new_pose[1], new_pose[2], current_pose[3], current_pose[4], current_pose[5]], a=1.2, v=0.0600)
    report_progress()
    set_digital_out(0, False)
    new_pose = pose_trans(tuft_coords, p[1.0737, 0.6962, 0.1500, 0, 0, 0])
    movel(p[new_pose[0], new_pose[1], new_pose[2], current_pose[3], current_pose[4], current_pose[5]], a=0.8, v=0.2000)
    report_progress()
    new_pose = pose_trans(tuft_coords, p[1.0757, 0.3578, 0.1500, 0, 0, 0])
    movel(p[new_pose[0], new_pose[1], new_pose[2], current_pose[3], current_pose[4], current_pose[5]], a=1.2, v=0.2000)
    report_progress()
    new_pose = pose_trans(tuft_coords, p[1.0757, 0.3578, -0.0020, 0, 0, 0])
    movel(p[new_pose[0], new_pose[1], new_pose[2], current_pose[3], current_pose[4], current_pose[5]], a=0.8, v=0.2000)
    report_progress()
    set_digital_out(0, True)
    new_pose = pose_trans(tuft_coords, p[1.0757, 0.6922, -0.0020, 0, 0, 0])
    movel(p[new_pose[0], new_pose[1], new_pose[2], current_pose[3], current_pose[4], current_pose[5]], a=1.2, v=0.0600)
    report_progress()
    set_digital_out(0, False)
    new_pose = pose_trans(tuft_coords, p[1.0757, 0.6922, 0.1500, 0, 0, 0])
    movel(p[new_pose[0], new_pose[1], new_pose[2], current_pose[3], current_pose[4], current_pose[5]], a=0.8, v=0.2000)
    report_progress()
    new_pose = pose_trans(tuft_coords, p[1.0776, 0.3617, 0.1500, 0, 0, 0])
    movel(p[new_pose[0], new_pose[1], new_pose[2], current_pose[3], current_pose[4], current_pose[5]], a=1.2, v=0.2000)
    report_progress()
    new_pose = pose_trans(tuft_coords, p[1.0776, 0.3617, -0.0020, 0, 0, 0])
    movel(p[new_pose[0], new_pose[1], new_pose[2], current_pose[3], current_pose[4], current_pose[5]], a=0.8, v=0.2000)
    report_progress()
    set_digital_out(0, True)
    new_pose = pose_trans(tuft_coords, p[1.0776, 0.6883, -0.0020, 0, 0, 0])
    movel(p[new_pose[0], new_pose[1], new_pose[2], current_pose[3], current_pose[4], current_pose[5]], a=1.2, v=0.0600)
    report_progress()
    set_digital_out(0, False)
    new_pose = pose_trans(tuft_coords, p[1.0776, 0.6883, 0.1500, 0, 0, 0])
    movel(p[new_pose[0], new_pose[1], new_pose[2], current_pose[3], current_pose[4], current_pose[5]], a=0.8, v=0.2000)
    report_progress()
    new_pose = pose_trans(tuft_coords, p[1.0796, 0.3657, 0.1500, 0, 0, 0])
    movel(p[new_pose[0], new_pose[1], new_pose[2], current_pose[3], current_pose[4], current_pose[5]], a=1.2, v=0.2000)
    report_progress()
    new_pose = pose_trans(tuft_coords, p[1.0796, 0.3657, -0.0020, 0, 0, 0])
    movel(p[new_pose[0], new_pose[1], new_pose[2], current_pose[3], current_pose[4], current_pose[5]], a=0.8, v=0.2000)
    report_progress()
    set_digital_out(0, True)
    new_pose = pose_trans(tuft_coords, p[1.0796, 0.6843, -0.0020, 0, 0, 0])
    movel(p[new_pose[0], new_pose[1], new_pose[2], current_pose[3], current_pose[4], current_pose[5]], a=1.2, v=0.0600)
    report_progress()
    set_digital_out(0, False)
    new_pose = pose_trans(tuft_coords, p[1.0796, 0.6843, 0.1500, 0, 0, 0])
    movel(p[new_pose[0], new_pose[1], new_pose[2], current_pose[3], current_pose[4], current_pose[5]], a=0.8, v=0.2000)
    report_progress()
    new_pose = pose_trans(tuft_coords, p[1.0815, 0.3696, 0.1500, 0, 0, 0])
    movel(p[new_pose[0], new_pose[1], new_pose[2], current_pose[3], current_pose[4], current_pose[5]], a=1.2, v=0.2000)
    report_progress()
    new_pose = pose_trans(tuft_coords, p[1.0815, 0.3696, -0.0020, 0, 0, 0])
    movel(p[new_pose[0], new_pose[1], new_pose[2], current_pose[3], current_pose[4], current_pose[5]], a=0.8, v=0.2000)
    report_progress()
    set_digital_out(0, True)
    new_pose = pose_trans(tuft_coords, p[1.0815, 0.6804, -0.0020, 0, 0, 0])
    movel(p[new_pose[0], new_pose[1], new_pose[2], current_pose[3], current_pose[4], current_pose[5]], a=1.2, v=0.0600)
    report_progress()
    set_digital_out(0, False)
    new_pose = pose_trans(tuft_coords, p[1.0815, 0.6804, 0.1500, 0, 0, 0])
    movel(p[new_pose[0], new_pose[1], new_pose[2], current_pose[3], current_pose[4], current_pose[5]], a=0.8, v=0.2000)
    report_progress()
    new_pose = pose_trans(tuft_coords, p[1.0835, 0.3736, 0.1500, 0, 0, 0])
    movel(p[new_pose[0], new_pose[1], new_pose[2], current_pose[3], current_pose[4], current_pose[5]], a=1.2, v=0.2000)
    report_progress()
    new_pose = pose_trans(tuft_coords, p[1.0835, 0.3736, -0.0020, 0, 0, 0])
    movel(p[new_pose[0], new_pose[1], new_pose[2], current_pose[3], current_pose[4], current_pose[5]], a=0.8, v=0.2000)
    report_progress()
    set_digital_out(0, True)
    new_pose = pose_trans(tuft_coords, p[1.0835, 0.6764, -0.0020, 0, 0, 0])
    movel(p[new_pose[0], new_pose[1], new_pose[2], current_pose[3], current_pose[4], current_pose[5]], a=1.2, v=0.0600)
    report_progress()
    set_digital_out(0, False)
    new_pose = pose_trans(tuft_coords, p[1.0835, 0.6764, 0.1500, 0, 0, 0])
    movel(p[new_pose[0], new_pose[1], new_pose[2], current_pose[3], current_pose[4], current_pose[5]], a=0.8, v=0.2000)
    report_progress()
    new_pose = pose_trans(tuft_coords, p[1.0854, 0.3795, 0.1500, 0, 0, 0])
    movel(p[new_pose[0], new_pose[1], new_pose[2], current_pose[3], current_pose[4], current_pose[5]], a=1.2, v=0.2000)
    report_progress()
    new_pose = pose_trans(tuft_coords, p[1.0854, 0.3795, -0.0020, 0, 0, 0])
    movel(p[new_pose[0], new_pose[1], new_pose[2], current_pose[3], current_pose[4], current_pose[5]], a=0.8, v=0.2000)
    report_progress()
    set_digital_out(0, True)
    new_pose = pose_trans(tuft_coords, p[1.0854, 0.6705, -0.0020, 0, 0, 0])
    movel(p[new_pose[0], new_pose[1], new_pose[2], current_pose[3], current_pose[4], current_pose[5]], a=1.2, v=0.0600)
    report_progress()
    set_digital_out(0, False)
    new_pose = pose_trans(tuft_coords, p[1.0854, 0.6705, 0.1500, 0, 0, 0])
    movel(p[new_pose[0], new_pose[1], new_pose[2], current_pose[3], current_pose[4], current_pose[5]], a=0.8, v=0.2000)
    report_progress()
    new_pose = pose_trans(tuft_coords, p[1.0874, 0.3835, 0.1500, 0, 0, 0])
    movel(p[new_pose[0], new_pose[1], new_pose[2], current_pose[3], current_pose[4], current_pose[5]], a=1.2, v=0.2000)
    report_progress()
    new_pose = pose_trans(tuft_coords, p[1.0874, 0.3835, -0.0020, 0, 0, 0])
    movel(p[new_pose[0], new_pose[1], new_pose[2], current_pose[3], current_pose[4], current_pose[5]], a=0.8, v=0.2000)
    report_progress()
    set_digital_out(0, True)
    new_pose = pose_trans(tuft_coords, p[1.0874, 0.6665, -0.0020, 0, 0, 0])
    movel(p[new_pose[0], new_pose[1], new_pose[2], current_pose[3], current_pose[4], current_pose[5]], a=1.2, v=0.0600)
    report_progress()
    set_digital_out(0, False)
    new_pose = pose_trans(tuft_coords, p[1.0874, 0.6665, 0.1500, 0, 0, 0])
    movel(p[new_pose[0], new_pose[1], new_pose[2], current_pose[3], current_pose[4], current_pose[5]], a=0.8, v=0.2000)
    report_progress()
    new_pose = pose_trans(tuft_coords, p[1.0893, 0.3874, 0.1500, 0, 0, 0])
    movel(p[new_pose[0], new_pose[1], new_pose[2], current_pose[3], current_pose[4], current_pose[5]], a=1.2, v=0.2000)
    report_progress()
    new_pose = pose_trans(tuft_coords, p[1.0893, 0.3874, -0.0020, 0, 0, 0])
    movel(p[new_pose[0], new_pose[1], new_pose[2], current_pose[3], current_pose[4], current_pose[5]], a=0.8, v=0.2000)
    report_progress()
    set_digital_out(0, True)
    new_pose = pose_trans(tuft_coords, p[1.0893, 0.6626, -0.0020, 0, 0, 0])
    movel(p[new_pose[0], new_pose[1], new_pose[2], current_pose[3], current_pose[4], current_pose[5]], a=1.2, v=0.0600)
    report_progress()
    set_digital_out(0, False)
    new_pose = pose_trans(tuft_coords, p[1.0893, 0.6626, 0.1500, 0, 0, 0])
    movel(p[new_pose[0], new_pose[1], new_pose[2], current_pose[3], current_pose[4], current_pose[5]], a=0.8, v=0.2000)
    report_progress()
    new_pose = pose_trans(tuft_coords, p[1.0913, 0.3934, 0.1500, 0, 0, 0])
    movel(p[new_pose[0], new_pose[1], new_pose[2], current_pose[3], current_pose[4], current_pose[5]], a=1.2, v=0.2000)
    report_progress()
    new_pose = pose_trans(tuft_coords, p[1.0913, 0.3934, -0.0020, 0, 0, 0])
    movel(p[new_pose[0], new_pose[1], new_pose[2], current_pose[3], current_pose[4], current_pose[5]], a=0.8, v=0.2000)
    report_progress()
    set_digital_out(0, True)
    new_pose = pose_trans(tuft_coords, p[1.0913, 0.6566, -0.0020, 0, 0, 0])
    movel(p[new_pose[0], new_pose[1], new_pose[2], current_pose[3], current_pose[4], current_pose[5]], a=1.2, v=0.0600)
    report_progress()
    set_digital_out(0, False)
    new_pose = pose_trans(tuft_coords, p[1.0913, 0.6566, 0.1500, 0, 0, 0])
    movel(p[new_pose[0], new_pose[1], new_pose[2], current_pose[3], current_pose[4], current_pose[5]], a=0.8, v=0.2000)
    report_progress()
    new_pose = pose_trans(tuft_coords, p[1.0932, 0.3993, 0.1500, 0, 0, 0])
    movel(p[new_pose[0], new_pose[1], new_pose[2], current_pose[3], current_pose[4], current_pose[5]], a=1.2, v=0.2000)
    report_progress()
    new_pose = pose_trans(tuft_coords, p[1.0932, 0.3993, -0.0020, 0, 0, 0])
    movel(p[new_pose[0], new_pose[1], new_pose[2], current_pose[3], current_pose[4], current_pose[5]], a=0.8, v=0.2000)
    report_progress()
    set_digital_out(0, True)
    new_pose = pose_trans(tuft_coords, p[1.0932, 0.6507, -0.0020, 0, 0, 0])
    movel(p[new_pose[0], new_pose[1], new_pose[2], current_pose[3], current_pose[4], current_pose[5]], a=1.2, v=0.0600)
    report_progress()
    set_digital_out(0, False)
    new_pose = pose_trans(tuft_coords, p[1.0932, 0.6507, 0.1500, 0, 0, 0])
    movel(p[new_pose[0], new_pose[1], new_pose[2], current_pose[3], current_pose[4], current_pose[5]], a=0.8, v=0.2000)
    report_progress()
    new_pose = pose_trans(tuft_coords, p[1.0951, 0.4053, 0.1500, 0, 0, 0])
    movel(p[new_pose[0], new_pose[1], new_pose[2], current_pose[3], current_pose[4], current_pose[5]], a=1.2, v=0.2000)
    report_progress()
    new_pose = pose_trans(tuft_coords, p[1.0951, 0.4053, -0.0020, 0, 0, 0])
    movel(p[new_pose[0], new_pose[1], new_pose[2], current_pose[3], current_pose[4], current_pose[5]], a=0.8, v=0.2000)
    report_progress()
    set_digital_out(0, True)
    new_pose = pose_trans(tuft_coords, p[1.0951, 0.6447, -0.0020, 0, 0, 0])
    movel(p[new_pose[0], new_pose[1], new_pose[2], current_pose[3], current_pose[4], current_pose[5]], a=1.2, v=0.0600)
    report_progress()
    set_digital_out(0, False)
    new_pose = pose_trans(tuft_coords, p[1.0951, 0.6447, 0.1500, 0, 0, 0])
    movel(p[new_pose[0], new_pose[1], new_pose[2], current_pose[3], current_pose[4], current_pose[5]], a=0.8, v=0.2000)
    report_progress()
    new_pose = pose_trans(tuft_coords, p[1.0971, 0.4092, 0.1500, 0, 0, 0])
    movel(p[new_pose[0], new_pose[1], new_pose[2], current_pose[3], current_pose[4], current_pose[5]], a=1.2, v=0.2000)
    report_progress()
    new_pose = pose_trans(tuft_coords, p[1.0971, 0.4092, -0.0020, 0, 0, 0])
    movel(p[new_pose[0], new_pose[1], new_pose[2], current_pose[3], current_pose[4], current_pose[5]], a=0.8, v=0.2000)
    report_progress()
    set_digital_out(0, True)
    new_pose = pose_trans(tuft_coords, p[1.0971, 0.6408, -0.0020, 0, 0, 0])
    movel(p[new_pose[0], new_pose[1], new_pose[2], current_pose[3], current_pose[4], current_pose[5]], a=1.2, v=0.0600)
    report_progress()
    set_digital_out(0, False)
    new_pose = pose_trans(tuft_coords, p[1.0971, 0.6408, 0.1500, 0, 0, 0])
    movel(p[new_pose[0], new_pose[1], new_pose[2], current_pose[3], current_pose[4], current_pose[5]], a=0.8, v=0.2000)
    report_progress()
    new_pose = pose_trans(tuft_coords, p[1.0990, 0.4171, 0.1500, 0, 0, 0])
    movel(p[new_pose[0], new_pose[1], new_pose[2], current_pose[3], current_pose[4], current_pose[5]], a=1.2, v=0.2000)
    report_progress()
    new_pose = pose_trans(tuft_coords, p[1.0990, 0.4171, -0.0020, 0, 0, 0])
    movel(p[new_pose[0], new_pose[1], new_pose[2], current_pose[3], current_pose[4], current_pose[5]], a=0.8, v=0.2000)
    report_progress()
    set_digital_out(0, True)
    new_pose = pose_trans(tuft_coords, p[1.0990, 0.6329, -0.0020, 0, 0, 0])
    movel(p[new_pose[0], new_pose[1], new_pose[2], current_pose[3], current_pose[4], current_pose[5]], a=1.2, v=0.0600)
    report_progress()
    set_digital_out(0, False)
    new_pose = pose_trans(tuft_coords, p[1.0990, 0.6329, 0.1500, 0, 0, 0])
    movel(p[new_pose[0], new_pose[1], new_pose[2], current_pose[3], current_pose[4], current_pose[5]], a=0.8, v=0.2000)
    report_progress()
    new_pose = pose_trans(tuft_coords, p[1.1010, 0.4231, 0.1500, 0, 0, 0])
    movel(p[new_pose[0], new_pose[1], new_pose[2], current_pose[3], current_pose[4], current_pose[5]], a=1.2, v=0.2000)
    report_progress()
    new_pose = pose_trans(tuft_coords, p[1.1010, 0.4231, -0.0020, 0, 0, 0])
    movel(p[new_pose[0], new_pose[1], new_pose[2], current_pose[3], current_pose[4], current_pose[5]], a=0.8, v=0.2000)
    report_progress()
    set_digital_out(0, True)
    new_pose = pose_trans(tuft_coords, p[1.1010, 0.6269, -0.0020, 0, 0, 0])
    movel(p[new_pose[0], new_pose[1], new_pose[2], current_pose[3], current_pose[4], current_pose[5]], a=1.2, v=0.0600)
    report_progress()
    set_digital_out(0, False)
    new_pose = pose_trans(tuft_coords, p[1.1010, 0.6269, 0.1500, 0, 0, 0])
    movel(p[new_pose[0], new_pose[1], new_pose[2], current_pose[3], current_pose[4], current_pose[5]], a=0.8, v=0.2000)
    report_progress()
    new_pose = pose_trans(tuft_coords, p[1.1029, 0.4310, 0.1500, 0, 0, 0])
    movel(p[new_pose[0], new_pose[1], new_pose[2], current_pose[3], current_pose[4], current_pose[5]], a=1.2, v=0.2000)
    report_progress()
    new_pose = pose_trans(tuft_coords, p[1.1029, 0.4310, -0.0020, 0, 0, 0])
    movel(p[new_pose[0], new_pose[1], new_pose[2], current_pose[3], current_pose[4], current_pose[5]], a=0.8, v=0.2000)
    report_progress()
    set_digital_out(0, True)
    new_pose = pose_trans(tuft_coords, p[1.1029, 0.6190, -0.0020, 0, 0, 0])
    movel(p[new_pose[0], new_pose[1], new_pose[2], current_pose[3], current_pose[4], current_pose[5]], a=1.2, v=0.0600)
    report_progress()
    set_digital_out(0, False)
    new_pose = pose_trans(tuft_coords, p[1.1029, 0.6190, 0.1500, 0, 0, 0])
    movel(p[new_pose[0], new_pose[1], new_pose[2], current_pose[3], current_pose[4], current_pose[5]], a=0.8, v=0.2000)
    report_progress()
    new_pose = pose_trans(tuft_coords, p[1.1049, 0.4389, 0.1500, 0, 0, 0])
    movel(p[new_pose[0], new_pose[1], new_pose[2], current_pose[3], current_pose[4], current_pose[5]], a=1.2, v=0.2000)
    report_progress()
    new_pose = pose_trans(tuft_coords, p[1.1049, 0.4389, -0.0020, 0, 0, 0])
    movel(p[new_pose[0], new_pose[1], new_pose[2], current_pose[3], current_pose[4], current_pose[5]], a=0.8, v=0.2000)
    report_progress()
    set_digital_out(0, True)
    new_pose = pose_trans(tuft_coords, p[1.1049, 0.6111, -0.0020, 0, 0, 0])
    movel(p[new_pose[0], new_pose[1], new_pose[2], current_pose[3], current_pose[4], current_pose[5]], a=1.2, v=0.0600)
    report_progress()
    set_digital_out(0, False)
    new_pose = pose_trans(tuft_coords, p[1.1049, 0.6111, 0.1500, 0, 0, 0])
    movel(p[new_pose[0], new_pose[1], new_pose[2], current_pose[3], current_pose[4], current_pose[5]], a=0.8, v=0.2000)
    report_progress()
    new_pose = pose_trans(tuft_coords, p[1.1068, 0.4468, 0.1500, 0, 0, 0])
    movel(p[new_pose[0], new_pose[1], new_pose[2], current_pose[3], current_pose[4], current_pose[5]], a=1.2, v=0.2000)
    report_progress()
    new_pose = pose_trans(tuft_coords, p[1.1068, 0.4468, -0.0020, 0, 0, 0])
    movel(p[new_pose[0], new_pose[1], new_pose[2], current_pose[3], current_pose[4], current_pose[5]], a=0.8, v=0.2000)
    report_progress()
    set_digital_out(0, True)
    new_pose = pose_trans(tuft_coords, p[1.1068, 0.6032, -0.0020, 0, 0, 0])
    movel(p[new_pose[0], new_pose[1], new_pose[2], current_pose[3], current_pose[4], current_pose[5]], a=1.2, v=0.0600)
    report_progress()
    set_digital_out(0, False)
    new_pose = pose_trans(tuft_coords, p[1.1068, 0.6032, 0.1500, 0, 0, 0])
    movel(p[new_pose[0], new_pose[1], new_pose[2], current_pose[3], current_pose[4], current_pose[5]], a=0.8, v=0.2000)
    report_progress()
    new_pose = pose_trans(tuft_coords, p[1.1087, 0.4567, 0.1500, 0, 0, 0])
    movel(p[new_pose[0], new_pose[1], new_pose[2], current_pose[3], current_pose[4], current_pose[5]], a=1.2, v=0.2000)
    report_progress()
    new_pose = pose_trans(tuft_coords, p[1.1087, 0.4567, -0.0020, 0, 0, 0])
    movel(p[new_pose[0], new_pose[1], new_pose[2], current_pose[3], current_pose[4], current_pose[5]], a=0.8, v=0.2000)
    report_progress()
    set_digital_out(0, True)
    new_pose = pose_trans(tuft_coords, p[1.1087, 0.5933, -0.0020, 0, 0, 0])
    movel(p[new_pose[0], new_pose[1], new_pose[2], current_pose[3], current_pose[4], current_pose[5]], a=1.2, v=0.0600)
    report_progress()
    set_digital_out(0, False)
    new_pose = pose_trans(tuft_coords, p[1.1087, 0.5933, 0.1500, 0, 0, 0])
    movel(p[new_pose[0], new_pose[1], new_pose[2], current_pose[3], current_pose[4], current_pose[5]], a=0.8, v=0.2000)
    report_progress()
    new_pose = pose_trans(tuft_coords, p[1.1107, 0.4686, 0.1500, 0, 0, 0])
    movel(p[new_pose[0], new_pose[1], new_pose[2], current_pose[3], current_pose[4], current_pose[5]], a=1.2, v=0.2000)
    report_progress()
    new_pose = pose_trans(tuft_coords, p[1.1107, 0.4686, -0.0020, 0, 0, 0])
    movel(p[new_pose[0], new_pose[1], new_pose[2], current_pose[3], current_pose[4], current_pose[5]], a=0.8, v=0.2000)
    report_progress()
    set_digital_out(0, True)
    new_pose = pose_trans(tuft_coords, p[1.1107, 0.5814, -0.0020, 0, 0, 0])
    movel(p[new_pose[0], new_pose[1], new_pose[2], current_pose[3], current_pose[4], current_pose[5]], a=1.2, v=0.0600)
    report_progress()
    set_digital_out(0, False)
    new_pose = pose_trans(tuft_coords, p[1.1107, 0.5814, 0.1500, 0, 0, 0])
    movel(p[new_pose[0], new_pose[1], new_pose[2], current_pose[3], current_pose[4], current_pose[5]], a=0.8, v=0.2000)
    report_progress()
    new_pose = pose_trans(tuft_coords, p[1.1126, 0.4824, 0.1500, 0, 0, 0])
    movel(p[new_pose[0], new_pose[1], new_pose[2], current_pose[3], current_pose[4], current_pose[5]], a=1.2, v=0.2000)
    report_progress()
    new_pose = pose_trans(tuft_coords, p[1.1126, 0.4824, -0.0020, 0, 0, 0])
    movel(p[new_pose[0], new_pose[1], new_pose[2], current_pose[3], current_pose[4], current_pose[5]], a=0.8, v=0.2000)
    report_progress()
    set_digital_out(0, True)
    new_pose = pose_trans(tuft_coords, p[1.1126, 0.5676, -0.0020, 0, 0, 0])
    movel(p[new_pose[0], new_pose[1], new_pose[2], current_pose[3], current_pose[4], current_pose[5]], a=1.2, v=0.0600)
    report_progress()
    set_digital_out(0, False)
    new_pose = pose_trans(tuft_coords, p[1.1126, 0.5676, 0.1500, 0, 0, 0])
    movel(p[new_pose[0], new_pose[1], new_pose[2], current_pose[3], current_pose[4], current_pose[5]], a=0.8, v=0.2000)
    report_progress()
    new_pose = pose_trans(tuft_coords, p[1.1146, 0.5062, 0.1500, 0, 0, 0])
    movel(p[new_pose[0], new_pose[1], new_pose[2], current_pose[3], current_pose[4], current_pose[5]], a=1.2, v=0.2000)
    report_progress()
    new_pose = pose_trans(tuft_coords, p[1.1146, 0.5062, -0.0020, 0, 0, 0])
    movel(p[new_pose[0], new_pose[1], new_pose[2], current_pose[3], current_pose[4], current_pose[5]], a=0.8, v=0.2000)
    report_progress()
    set_digital_out(0, True)
    new_pose = pose_trans(tuft_coords, p[1.1146, 0.5438, -0.0020, 0, 0, 0])
    movel(p[new_pose[0], new_pose[1], new_pose[2], current_pose[3], current_pose[4], current_pose[5]], a=1.2, v=0.0600)
    report_progress()
    set_digital_out(0, False)
    new_pose = pose_trans(tuft_coords, p[1.1146, 0.5438, 0.1500, 0, 0, 0])
    movel(p[new_pose[0], new_pose[1], new_pose[2], current_pose[3], current_pose[4], current_pose[5]], a=0.8, v=0.2000)
    report_progress()
    textmsg("Tufting job finished")
end
